(* Logix 5000 project; controller Explicit_Messaging vendor 1 type 14 code 192 rev 33.11; software revision 33.01 *)

TASK MainTask (continuous, watchdog 500 ms) : MainProgram, Robot_IO

MODULES
   Local : vendor 1 type 14 code 192 (5069 0, rev 33.11)
      R1 : vendor 356 type 12 code 2 (Ethernet 192.169.1.20, rev 2.1, StandardDataDriven RPI 32 ms)
END_MODULES

TYPE Robot_Fanuc :
STRUCT
   i : Robot_Fanuc_PLC_Inputs;
   o : Robot_Fanuc_PLC_Outputs;
   Ctrl : Robot_Fanuc_Ctrl;
   Proc : Robot_Fanuc_Process;
END_STRUCT
END_TYPE

TYPE Robot_Fanuc_Ctrl :
STRUCT
   GI_1 : SINT;   // GI[1]
   GO_1 : SINT;   // GO[1]
END_STRUCT
END_TYPE

TYPE Robot_Fanuc_PLC_Inputs :
STRUCT
   UO01_CmdEnbl : BOOL;   // UO 1 CMD Enabled
   UO02_SysRdy : BOOL;   // UO 2 System Ready
   UO03_ProgRun : BOOL;   // UO 3 Program Running
   UO04_Paused : BOOL;   // UO 4 Program Paused
   UO05_Held : BOOL;   // UO 5 Motion Held
   UO06_Fault : BOOL;   // UO 6 Fault
   UO07_AtHome : BOOL;   // UO 7 At Perch
   UO08_TPEnbld : BOOL;   // UO 8 TP Enabled
   UO09_BattAlrm : BOOL;   // UO 9 Batt Alarm
   UO10_Busy : BOOL;   // UO 10 Busy
   UO11_PNS01Echo : BOOL;   // UO 11 PNS Acknowledge 1
   UO12_PNS02Echo : BOOL;   // UO 12 PNS Acknowledge 2
   UO13_PNS03Echo : BOOL;   // UO 13 PNS Acknowledge 3
   UO14_PNS04Echo : BOOL;   // UO 14 PNS Acknowledge 4
   UO15_PNS05Echo : BOOL;   // UO 15 PNS Acknowledge 5
   UO16_PNS06Echo : BOOL;   // UO 16 PNS Acknowledge 6
   UO17_PNS07Echo : BOOL;   // UO 17 PNS Acknowledge 7
   UO18_PNS08Echo : BOOL;   // UO 18 PNS Acknowledge 8
   UO19_Snack : BOOL;   // UO 19 Snack
   UO20_Reserved : BOOL;   // UO 20 Reserved
   DO021 : BOOL;
   DO022 : BOOL;
   DO023 : BOOL;
   DO024 : BOOL;
   DO025 : BOOL;
   DO026 : BOOL;
   DO027 : BOOL;
   DO028 : BOOL;
   DO029 : BOOL;
   DO030 : BOOL;
   DO031 : BOOL;
   DO032 : BOOL;
   DO033 : BOOL;
   DO034 : BOOL;
   DO035 : BOOL;
   DO036 : BOOL;
   DO037 : BOOL;
   DO038 : BOOL;
   DO039 : BOOL;
   DO040 : BOOL;
   DO041 : BOOL;
   DO042 : BOOL;
   DO043 : BOOL;
   DO044 : BOOL;
   DO045 : BOOL;
   DO046 : BOOL;
   DO047 : BOOL;
   DO048 : BOOL;
   DO049 : BOOL;
   DO050 : BOOL;
   DO051 : BOOL;
   DO052 : BOOL;
   DO053 : BOOL;
   DO054 : BOOL;
   DO055 : BOOL;
   DO056 : BOOL;
   DO057 : BOOL;
   DO058 : BOOL;
   DO059 : BOOL;
   DO060 : BOOL;
   DO061 : BOOL;
   DO062 : BOOL;
   DO063 : BOOL;
   DO064 : BOOL;
   DO065 : BOOL;
   DO066 : BOOL;
   DO067 : BOOL;
   DO068 : BOOL;
   DO069 : BOOL;
   DO070 : BOOL;
   DO071 : BOOL;
   DO072 : BOOL;
   DO073 : BOOL;
   DO074 : BOOL;
   DO075 : BOOL;
   DO076 : BOOL;
   DO077 : BOOL;
   DO078 : BOOL;
   DO079 : BOOL;
   DO080 : BOOL;
   DO081 : BOOL;
   DO082 : BOOL;
   DO083 : BOOL;
   DO084 : BOOL;
   DO085 : BOOL;
   DO086 : BOOL;
   DO087 : BOOL;
   DO088 : BOOL;
   DO089 : BOOL;
   DO090 : BOOL;
   DO091 : BOOL;
   DO092 : BOOL;
   DO093 : BOOL;
   DO094 : BOOL;
   DO095 : BOOL;
   DO096 : BOOL;
   DO097 : BOOL;
   DO099 : BOOL;
   DO100 : BOOL;
   DO101 : BOOL;
   DO102 : BOOL;
   DO103 : BOOL;
   DO104 : BOOL;
   DO105 : BOOL;
   DO106 : BOOL;
   DO107 : BOOL;
   DO108 : BOOL;
   DO109 : BOOL;
   DO110 : BOOL;
   DO111 : BOOL;
   DO112 : BOOL;
   DO113 : BOOL;
   DO114 : BOOL;
   DO115 : BOOL;
   DO116 : BOOL;
   DO117 : BOOL;
   DO118 : BOOL;
   DO119 : BOOL;
   DO120 : BOOL;
   DO121 : BOOL;
   DO122 : BOOL;
   DO123 : BOOL;
   DO124 : BOOL;
   DO125 : BOOL;
   DO126 : BOOL;
   DO127 : BOOL;
   DO128 : BOOL;
   DO129 : BOOL;
   DO130 : BOOL;
   DO131 : BOOL;
   DO132 : BOOL;
   DO133 : BOOL;
   DO134 : BOOL;
   DO135 : BOOL;
   DO136 : BOOL;
   DO137 : BOOL;
   DO138 : BOOL;
   DO139 : BOOL;
   DO140 : BOOL;
   DO141 : BOOL;
   DO142 : BOOL;
   DO143 : BOOL;
   DO144 : BOOL;
   DO145 : BOOL;
   DO146 : BOOL;
   DO147 : BOOL;
   DO148 : BOOL;
   DO149 : BOOL;
   DO150 : BOOL;
   DO151 : BOOL;
   DO152 : BOOL;
   DO153 : BOOL;
   DO154 : BOOL;
   DO155 : BOOL;
   DO156 : BOOL;
   DO157 : BOOL;
   DO158 : BOOL;
   DO159 : BOOL;
   DO160 : BOOL;
   DO161 : BOOL;
   DO162 : BOOL;
   DO163 : BOOL;
   DO164 : BOOL;
   DO165 : BOOL;
   DO166 : BOOL;
   DO167 : BOOL;
   DO168 : BOOL;
   DO169 : BOOL;
   DO170 : BOOL;
   DO171 : BOOL;
   DO172 : BOOL;
   DO173 : BOOL;
   DO174 : BOOL;
   DO175 : BOOL;
   DO176 : BOOL;
   DO177 : BOOL;
   DO178 : BOOL;
   DO179 : BOOL;
   DO180 : BOOL;
   DO181 : BOOL;
   DO182 : BOOL;
   DO183 : BOOL;
   DO184 : BOOL;
   DO185 : BOOL;
   DO186 : BOOL;
   DO187 : BOOL;
   DO188 : BOOL;
   DO189 : BOOL;
   DO190 : BOOL;
   DO191 : BOOL;
   DO192 : BOOL;
   DO193 : BOOL;
   DO194 : BOOL;
   DO195 : BOOL;
   DO196 : BOOL;
   DO197 : BOOL;
   DO198 : BOOL;
   DO199 : BOOL;
   DO200 : BOOL;
   DO201 : BOOL;
   DO202 : BOOL;
   DO203 : BOOL;
   DO204 : BOOL;
   DO205 : BOOL;
   DO206 : BOOL;
   DO207 : BOOL;
   DO208 : BOOL;
   DO209 : BOOL;
   DO210 : BOOL;
   DO211 : BOOL;
   DO212 : BOOL;
   DO213 : BOOL;
   DO214 : BOOL;
   DO215 : BOOL;
   DO216 : BOOL;
   DO217 : BOOL;
   DO218 : BOOL;
   DO219 : BOOL;
   DO220 : BOOL;
   DO221 : BOOL;
   DO222 : BOOL;
   DO223 : BOOL;
   DO224 : BOOL;
   DO225 : BOOL;
   DO226 : BOOL;
   DO227 : BOOL;
   DO228 : BOOL;
   DO229 : BOOL;
   DO230 : BOOL;
   DO231 : BOOL;
   DO232 : BOOL;
   DO233 : BOOL;
   DO234 : BOOL;
   DO235 : BOOL;
   DO236 : BOOL;
   DO237 : BOOL;
   DO238 : BOOL;
   DO239 : BOOL;
   DO240 : BOOL;
   DO241 : BOOL;
   DO242 : BOOL;
   DO243 : BOOL;
   DO244 : BOOL;
   DO245 : BOOL;
   DO246 : BOOL;
   DO247 : BOOL;
   DO248 : BOOL;
   DO249 : BOOL;
   DO250 : BOOL;
   DO251 : BOOL;
   DO252 : BOOL;
   DO253 : BOOL;
   DO254 : BOOL;
   DO255 : BOOL;
   DO256 : BOOL;
END_STRUCT
END_TYPE

TYPE Robot_Fanuc_PLC_Outputs :
STRUCT
   UI01_ImStp : BOOL;   // UI 1 IMSTP
   UI02_Hold : BOOL;   // UI 2 Hold
   UI03_SafeSpeed : BOOL;   // UI 3 SFSPD
   UI04_CstopI : BOOL;   // UI 4 Cycle Stop
   UI05_FaultReset : BOOL;   // UI 5 Fault Reset
   UI06_Start : BOOL;   // UI 6 Start
   UI07_Home : BOOL;   // UI 7 Home
   UI08_Enable : BOOL;   // UI 8 Enable
   UI09_PNS01 : BOOL;   // UI 9 PNS 1
   UI10_PNS02 : BOOL;   // UI 10 PNS 2
   UI11_PNS03 : BOOL;   // UI 11 PNS 3
   UI12_PNS04 : BOOL;   // UI 12 PNS 4
   UI13_PNS05 : BOOL;   // UI 13 PNS 5
   UI14_PNS06 : BOOL;   // UI 14 PNS 6
   UI15_PNS07 : BOOL;   // UI 15 PNS 7
   UI16_PNS08 : BOOL;   // UI 16 PNS 8
   UI17_PNSStrobe : BOOL;   // UI 17 PNS Strobe
   UI18_ProdStart : BOOL;   // UI 18 PNS Product Start
   DI019 : BOOL;
   DI020 : BOOL;
   DI021 : BOOL;
   DI022 : BOOL;
   DI023 : BOOL;
   DI024 : BOOL;
   DI025 : BOOL;
   DI026 : BOOL;
   DI027 : BOOL;
   DI028 : BOOL;
   DI029 : BOOL;
   DI030 : BOOL;
   DI031 : BOOL;
   DI032 : BOOL;
   DI033 : BOOL;
   DI034 : BOOL;
   DI035 : BOOL;
   DI036 : BOOL;
   DI037 : BOOL;
   DI038 : BOOL;
   DI039 : BOOL;
   DI040 : BOOL;
   DI041 : BOOL;
   DI042 : BOOL;
   DI043 : BOOL;
   DI044 : BOOL;
   DI045 : BOOL;
   DI046 : BOOL;
   DI047 : BOOL;
   DI048 : BOOL;
   DI049 : BOOL;
   DI050 : BOOL;
   DI051 : BOOL;
   DI052 : BOOL;
   DI053 : BOOL;
   DI054 : BOOL;
   DI055 : BOOL;
   DI056 : BOOL;
   DI057 : BOOL;
   DI058 : BOOL;
   DI059 : BOOL;
   DI060 : BOOL;
   DI061 : BOOL;
   DI062 : BOOL;
   DI063 : BOOL;
   DI064 : BOOL;
   DI065 : BOOL;
   DI066 : BOOL;
   DI067 : BOOL;
   DI068 : BOOL;
   DI069 : BOOL;
   DI070 : BOOL;
   DI071 : BOOL;
   DI072 : BOOL;
   DI073 : BOOL;
   DI074 : BOOL;
   DI075 : BOOL;
   DI076 : BOOL;
   DI077 : BOOL;
   DI078 : BOOL;
   DI079 : BOOL;
   DI080 : BOOL;
   DI081 : BOOL;
   DI082 : BOOL;
   DI083 : BOOL;
   DI084 : BOOL;
   DI085 : BOOL;
   DI086 : BOOL;
   DI087 : BOOL;
   DI088 : BOOL;
   DI089 : BOOL;
   DI090 : BOOL;
   DI091 : BOOL;
   DI092 : BOOL;
   DI093 : BOOL;
   DI094 : BOOL;
   DI095 : BOOL;
   DI096 : BOOL;
   DI097 : BOOL;
   DI098 : BOOL;
   DI099 : BOOL;
   DI100 : BOOL;
   DI101 : BOOL;
   DI102 : BOOL;
   DI103 : BOOL;
   DI104 : BOOL;
   DI105 : BOOL;
   DI106 : BOOL;
   DI107 : BOOL;
   DI108 : BOOL;
   DI109 : BOOL;
   DI110 : BOOL;
   DI111 : BOOL;
   DI112 : BOOL;
   DI113 : BOOL;
   DI114 : BOOL;
   DI115 : BOOL;
   DI116 : BOOL;
   DI117 : BOOL;
   DI118 : BOOL;
   DI119 : BOOL;
   DI120 : BOOL;
   DI121 : BOOL;
   DI122 : BOOL;
   DI123 : BOOL;
   DI124 : BOOL;
   DI125 : BOOL;
   DI126 : BOOL;
   DI127 : BOOL;
   DI128 : BOOL;
   DI129 : BOOL;
   DI130 : BOOL;
   DI131 : BOOL;
   DI132 : BOOL;
   DI133 : BOOL;
   DI134 : BOOL;
   DI135 : BOOL;
   DI136 : BOOL;
   DI137 : BOOL;
   DI138 : BOOL;
   DI139 : BOOL;
   DI140 : BOOL;
   DI141 : BOOL;
   DI142 : BOOL;
   DI143 : BOOL;
   DI144 : BOOL;
   DI145 : BOOL;
   DI146 : BOOL;
   DI147 : BOOL;
   DI148 : BOOL;
   DI149 : BOOL;
   DI150 : BOOL;
   DI151 : BOOL;
   DI152 : BOOL;
   DI153 : BOOL;
   DI154 : BOOL;
   DI155 : BOOL;
   DI156 : BOOL;
   DI157 : BOOL;
   DI158 : BOOL;
   DI159 : BOOL;
   DI160 : BOOL;
   DI161 : BOOL;
   DI162 : BOOL;
   DI163 : BOOL;
   DI164 : BOOL;
   DI165 : BOOL;
   DI166 : BOOL;
   DI167 : BOOL;
   DI168 : BOOL;
   DI169 : BOOL;
   DI170 : BOOL;
   DI171 : BOOL;
   DI172 : BOOL;
   DI173 : BOOL;
   DI174 : BOOL;
   DI175 : BOOL;
   DI176 : BOOL;
   DI177 : BOOL;
   DI178 : BOOL;
   DI179 : BOOL;
   DI180 : BOOL;
   DI181 : BOOL;
   DI182 : BOOL;
   DI183 : BOOL;
   DI184 : BOOL;
   DI185 : BOOL;
   DI186 : BOOL;
   DI187 : BOOL;
   DI188 : BOOL;
   DI189 : BOOL;
   DI190 : BOOL;
   DI191 : BOOL;
   DI192 : BOOL;
   DI193 : BOOL;
   DI194 : BOOL;
   DI195 : BOOL;
   DI196 : BOOL;
   DI197 : BOOL;
   DI198 : BOOL;
   DI199 : BOOL;
   DI200 : BOOL;
   DI201 : BOOL;
   DI202 : BOOL;
   DI203 : BOOL;
   DI204 : BOOL;
   DI205 : BOOL;
   DI206 : BOOL;
   DI207 : BOOL;
   DI208 : BOOL;
   DI209 : BOOL;
   DI210 : BOOL;
   DI211 : BOOL;
   DI212 : BOOL;
   DI213 : BOOL;
   DI214 : BOOL;
   DI215 : BOOL;
   DI216 : BOOL;
   DI217 : BOOL;
   DI218 : BOOL;
   DI219 : BOOL;
   DI220 : BOOL;
   DI221 : BOOL;
   DI222 : BOOL;
   DI223 : BOOL;
   DI224 : BOOL;
   DI225 : BOOL;
   DI226 : BOOL;
   DI227 : BOOL;
   DI228 : BOOL;
   DI229 : BOOL;
   DI230 : BOOL;
   DI231 : BOOL;
   DI232 : BOOL;
   DI233 : BOOL;
   DI234 : BOOL;
   DI235 : BOOL;
   DI236 : BOOL;
   DI237 : BOOL;
   DI238 : BOOL;
   DI239 : BOOL;
   DI240 : BOOL;
   DI241 : BOOL;
   DI242 : BOOL;
   DI243 : BOOL;
   DI244 : BOOL;
   DI245 : BOOL;
   DI246 : BOOL;
   DI247 : BOOL;
   DI248 : BOOL;
   DI249 : BOOL;
   DI250 : BOOL;
   DI251 : BOOL;
   DI252 : BOOL;
   DI253 : BOOL;
   DI254 : BOOL;
   DI255 : BOOL;
   DI256 : BOOL;
END_STRUCT
END_TYPE

TYPE Robot_Fanuc_Process :
STRUCT
   Data_Reg20 : Robot_MSG_Register;
END_STRUCT
END_TYPE

TYPE Robot_MSG_Register :
STRUCT
   Read_Delay : TIMER;
   Write_Delay : TIMER;
   Data_Read : REAL[10];
   Data_Write : REAL[10];
   Data_Match : BOOL;   // Data Match
   Data_Write_Save_PB : BOOL;   // Save PB
END_STRUCT
END_TYPE

TYPE STRING_088 :
STRUCT
   LEN : DINT;
   DATA : SINT[88];
END_STRUCT
END_TYPE

VAR_GLOBAL   (* controller tags *)
   Alarms : DINT;
   Empty_STR88 : STRING_088;
   R1_MSG_Registers : Robot_MSG_Register;
   Robot : Robot_Fanuc := (i.UO06_Fault := 1, Proc.Data_Reg20.Read_Delay.PRE := 1000, Proc.Data_Reg20.Write_Delay.PRE := 1000);
   Robot_Alarm_STR88 : STRING_088 := 'SRVO-003 Deadman switch released                                               ';
   Robot_MSG_Alarm : MESSAGE;
        MessageParameters(ServiceCode := 16#000e, DestinationTag := Robot_Alarm_STR88, ...)
   Robot_MSG_Alarm_Read_Delay : TIMER := (PRE := 1000, ACC := 491, EN := 1, TT := 1);
   Robot_MSG_Reg20_Read : MESSAGE;
        MessageParameters(ServiceCode := 16#0032, DestinationTag := R1_MSG_Registers.Data_Read[0], ...)
   Robot_MSG_Reg20_Write : MESSAGE;
        MessageParameters(ServiceCode := 16#0033, LocalElement := R1_MSG_Registers.Data_Write[0], ...)
END_VAR

PROGRAM MainProgram   (* main routine MainRoutine *)
VAR
   ONS : DINT;   // One Shot
END_VAR

ROUTINE Alarms   (* ladder *)
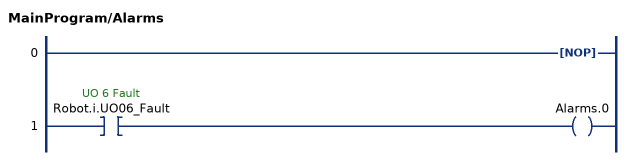
   0: NOP();
   1: XIC(Robot.i.UO06_Fault)OTE(Alarms.0);
END_ROUTINE

ROUTINE MainRoutine   (* ladder *)
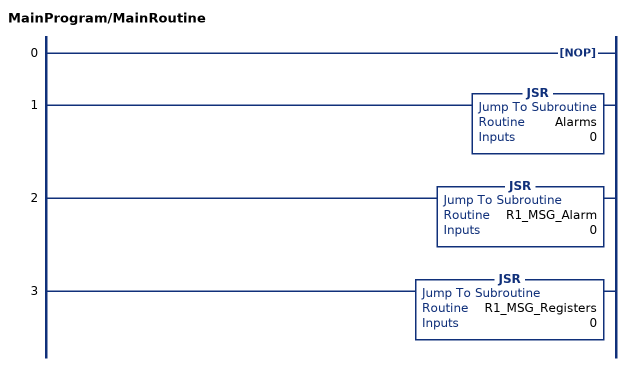
   0: NOP();
   1: JSR(Alarms,0);
   2: JSR(R1_MSG_Alarm,0);
   3: JSR(R1_MSG_Registers,0);
END_ROUTINE

ROUTINE R1_MSG_Alarm   (* ladder *)
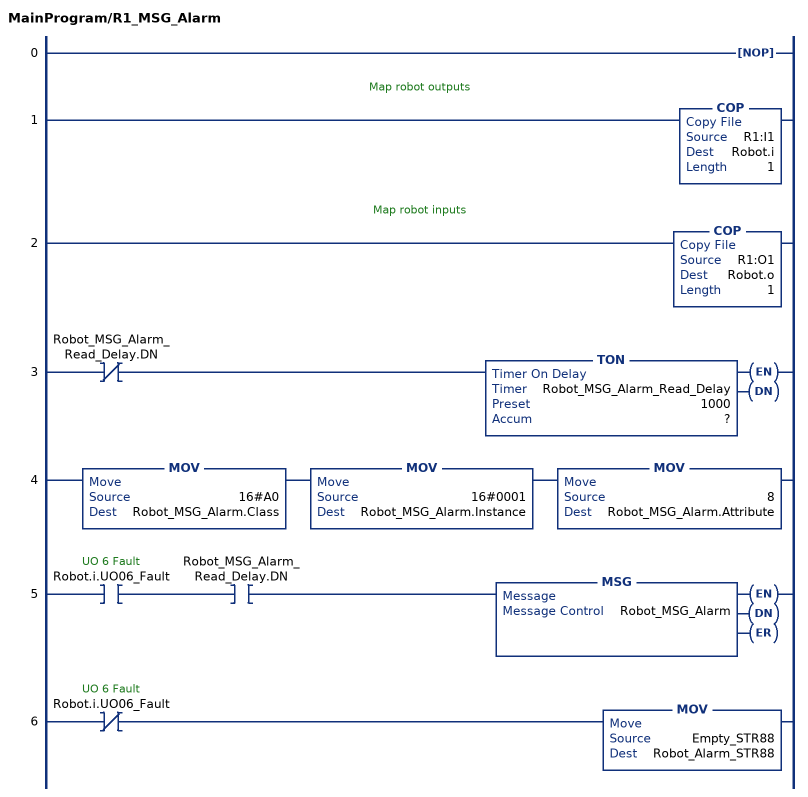
   0: NOP();
   // Map robot outputs
   1: COP(R1:I1,Robot.i,1);
   // Map robot inputs
   2: COP(R1:O1,Robot.o,1);
   3: XIO(Robot_MSG_Alarm_Read_Delay.DN)TON(Robot_MSG_Alarm_Read_Delay,?,?);
   4: MOV(16#A0,Robot_MSG_Alarm.Class)MOV(16#0001,Robot_MSG_Alarm.Instance)MOV(8,Robot_MSG_Alarm.Attribute);
   5: XIC(Robot.i.UO06_Fault)XIC(Robot_MSG_Alarm_Read_Delay.DN)MSG(Robot_MSG_Alarm);
   6: XIO(Robot.i.UO06_Fault)MOV(Empty_STR88,Robot_Alarm_STR88);
END_ROUTINE

ROUTINE R1_MSG_Registers   (* ladder *)
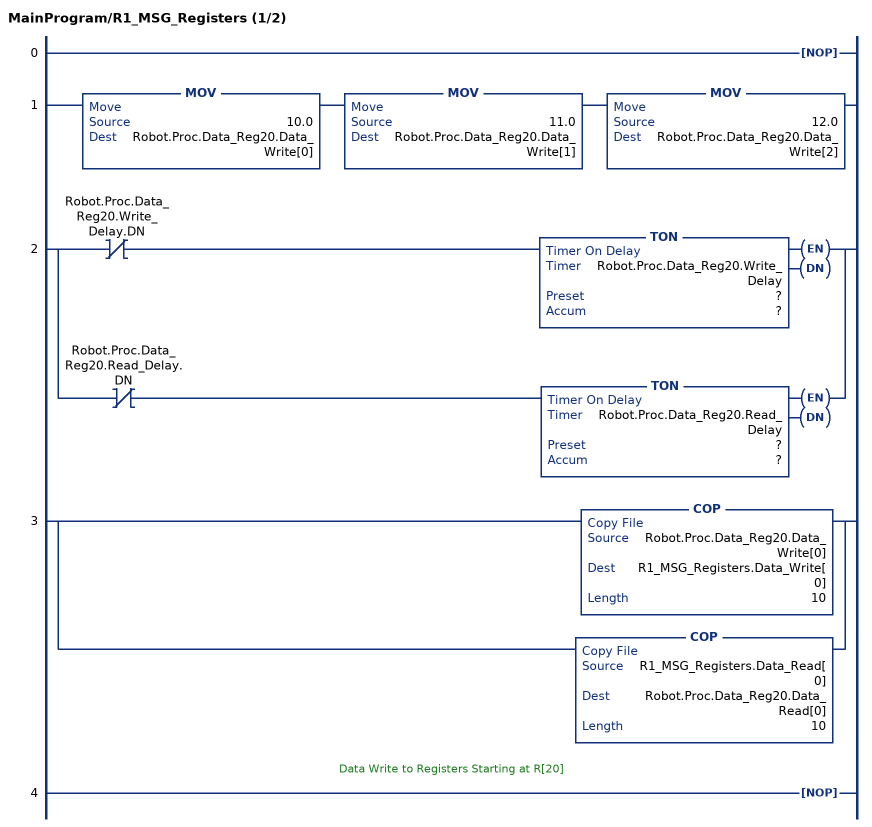
   0: NOP();
   1: MOV(10.0,Robot.Proc.Data_Reg20.Data_Write[0])MOV(11.0,Robot.Proc.Data_Reg20.Data_Write[1])MOV(12.0,Robot.Proc.Data_Reg20.Data_Write[2]);
   2: [XIO(Robot.Proc.Data_Reg20.Write_Delay.DN) TON(Robot.Proc.Data_Reg20.Write_Delay,?,?) ,XIO(Robot.Proc.Data_Reg20.Read_Delay.DN) TON(Robot.Proc.Data_Reg20.Read_Delay,?,?) ];
   3: [COP(Robot.Proc.Data_Reg20.Data_Write[0],R1_MSG_Registers.Data_Write[0],10) ,COP(R1_MSG_Registers.Data_Read[0],Robot.Proc.Data_Reg20.Data_Read[0],10) ];
   // Data Write to Registers Starting at R[20]
   4: NOP();
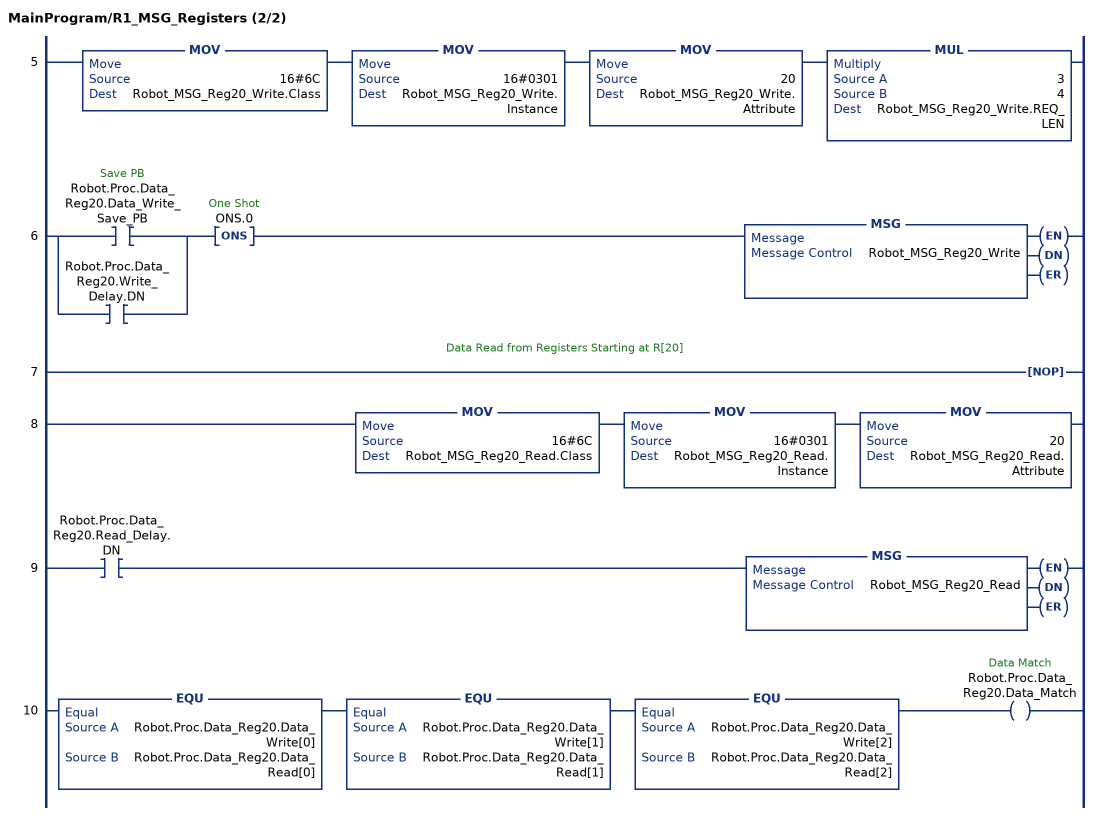
   5: MOV(16#6C,Robot_MSG_Reg20_Write.Class)MOV(16#0301,Robot_MSG_Reg20_Write.Instance)MOV(20,Robot_MSG_Reg20_Write.Attribute)MUL(3,4,Robot_MSG_Reg20_Write.REQ_LEN);
   6: [XIC(Robot.Proc.Data_Reg20.Data_Write_Save_PB) ,XIC(Robot.Proc.Data_Reg20.Write_Delay.DN) ]ONS(ONS.0)MSG(Robot_MSG_Reg20_Write);
   // Data Read from Registers Starting at R[20]
   7: NOP();
   8: MOV(16#6C,Robot_MSG_Reg20_Read.Class)MOV(16#0301,Robot_MSG_Reg20_Read.Instance)MOV(20,Robot_MSG_Reg20_Read.Attribute);
   9: XIC(Robot.Proc.Data_Reg20.Read_Delay.DN)MSG(Robot_MSG_Reg20_Read);
   10: EQU(Robot.Proc.Data_Reg20.Data_Write[0],Robot.Proc.Data_Reg20.Data_Read[0])EQU(Robot.Proc.Data_Reg20.Data_Write[1],Robot.Proc.Data_Reg20.Data_Read[1])EQU(Robot.Proc.Data_Reg20.Data_Write[2],Robot.Proc.Data_Reg20.Data_Read[2])OTE(Robot.Proc.Data_Reg20.Data_Match);
END_ROUTINE
END_PROGRAM

PROGRAM Robot_IO   (* main routine MainRoutine *)

ROUTINE MainRoutine   (* ladder *)
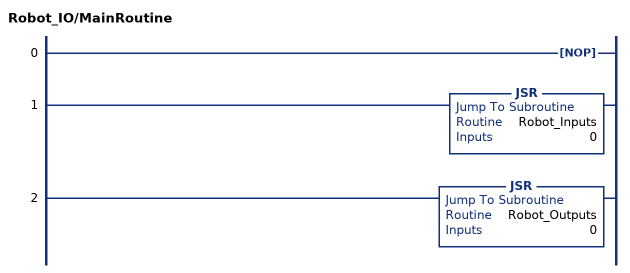
   0: NOP();
   1: JSR(Robot_Inputs,0);
   2: JSR(Robot_Outputs,0);
END_ROUTINE

ROUTINE Robot_Inputs   (* ladder *)
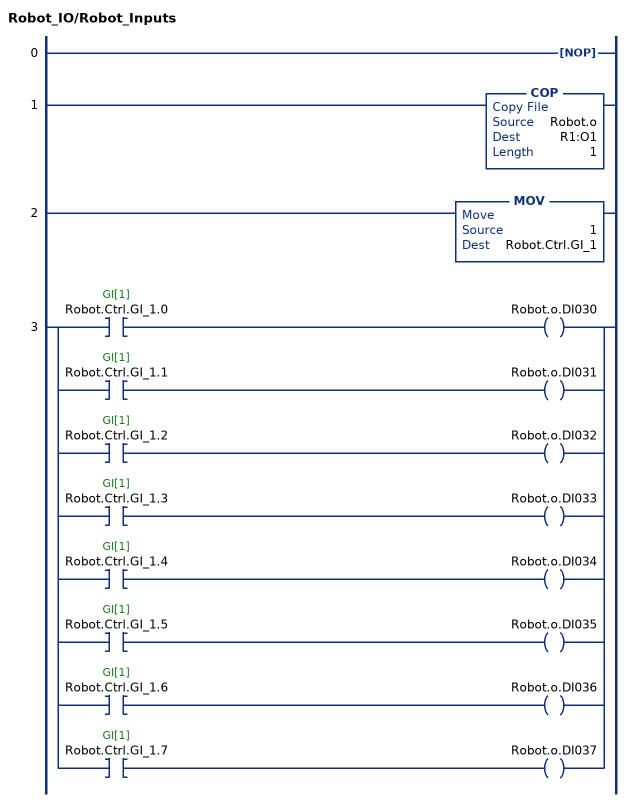
   0: NOP();
   1: COP(Robot.o,R1:O1,1);
   2: MOV(1,Robot.Ctrl.GI_1);
   3: [XIC(Robot.Ctrl.GI_1.0) OTE(Robot.o.DI030) ,XIC(Robot.Ctrl.GI_1.1) OTE(Robot.o.DI031) ,XIC(Robot.Ctrl.GI_1.2) OTE(Robot.o.DI032) ,XIC(Robot.Ctrl.GI_1.3) OTE(Robot.o.DI033) ,XIC(Robot.Ctrl.GI_1.4) OTE(Robot.o.DI034) ,XIC(Robot.Ctrl.GI_1.5) OTE(Robot.o.DI035) ,XIC(Robot.Ctrl.GI_1.6) OTE(Robot.o.DI036) ,XIC(Robot.Ctrl.GI_1.7) OTE(Robot.o.DI037) ];
END_ROUTINE

ROUTINE Robot_Outputs   (* ladder *)
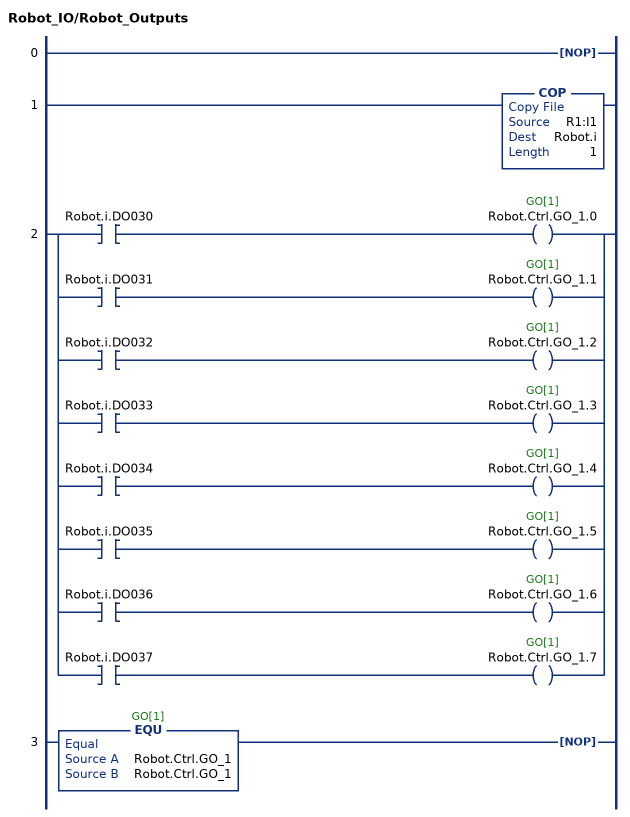
   0: NOP();
   1: COP(R1:I1,Robot.i,1);
   2: [XIC(Robot.i.DO030) OTE(Robot.Ctrl.GO_1.0) ,XIC(Robot.i.DO031) OTE(Robot.Ctrl.GO_1.1) ,XIC(Robot.i.DO032) OTE(Robot.Ctrl.GO_1.2) ,XIC(Robot.i.DO033) OTE(Robot.Ctrl.GO_1.3) ,XIC(Robot.i.DO034) OTE(Robot.Ctrl.GO_1.4) ,XIC(Robot.i.DO035) OTE(Robot.Ctrl.GO_1.5) ,XIC(Robot.i.DO036) OTE(Robot.Ctrl.GO_1.6) ,XIC(Robot.i.DO037) OTE(Robot.Ctrl.GO_1.7) ];
   3: EQU(Robot.Ctrl.GO_1,Robot.Ctrl.GO_1)NOP();
END_ROUTINE
END_PROGRAM
